# EPICS substitutions: ek9000App/Db/EL3074.substitutions
file EL3074.template
{       pattern
        {
                TERMINAL,

        }
        {
        }
}
